// TIA Portal V20 export
DATA_BLOCK "BK30"   // DB237
// stored: MemoryReserve 100
   VAR
      "X10-1.SUCTION PAD TOP TAPE VACUUM ON" : Bool := FALSE;
      "X10-2.SUCTION PAD TOP TAPE VACUUM OFF" : Bool := FALSE;
      "X12-1.SUCTION PAD BTM TAPE VACUUM ON" : Bool := FALSE;
      "X12-2.SUCTION PAD BTM TAPE VACUUM OFF" : Bool := FALSE;
      "X14-1.STACK TABLE VACUUM ON" : Bool := FALSE;
      "X14-2.STACK TABLE VACUUM OFF" : Bool := FALSE;
      "X16-1.SPARE" : Bool := FALSE;
      "X16-2.SPARE" : Bool := FALSE;
   END_VAR
BEGIN
END_DATA_BLOCK
